% RSLogix 500 project FIVE_CONVEYER_SYS_BAK010.RSS, saved by version 8.30.00.16 %
PROJECT "UNTITLED"    % processor: Bul.1763 MicroLogix 1100 Series B %

PROGRAM FILES
  LAD 2   11 rungs
  LAD 3 "BELT 1"  5 rungs
  LAD 4 "BELT 2"  5 rungs
  LAD 5 "BELT 3"  5 rungs
  LAD 6 "BELT 4"  5 rungs
  LAD 7 "BELT 5"  5 rungs
  LAD 8 "SEQUENCING"  7 rungs

DATA FILES
  O0 OUTPUT  4 elements
  I1 INPUT  6 elements
  S2 STATUS  66 elements
  B3 BINARY  10 elements
  T4 TIMER  20 elements
  C5 COUNTER  1 elements
  R6 CONTROL  1 elements
  N7 INTEGER  1 elements
  F8 FLOAT  1 elements

LADDER 2
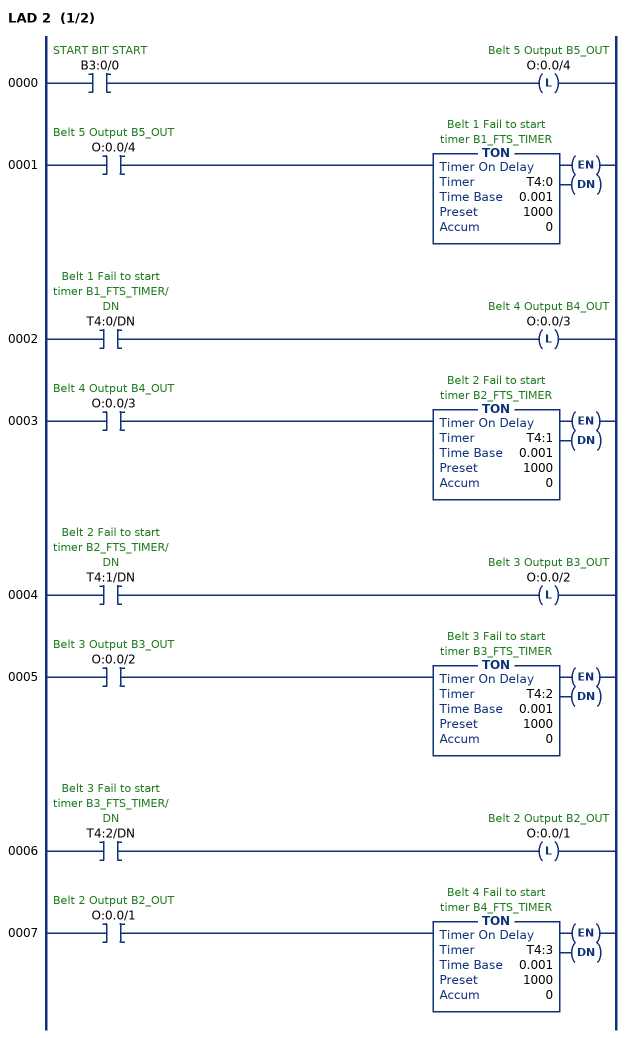
% Rung: 0 %  % edit flag set %
SOR XIC B3:0/0 OTL O:0.0/4 EOR
%   B3:0/0  START  "START BIT" %
%   O:0.0/4  B5_OUT  "Belt 5 Output" %
% Rung: 1 %  % edit flag set %
SOR XIC O:0.0/4 TON T4:0 0.001 1000 0 EOR
%   O:0.0/4  B5_OUT  "Belt 5 Output" %
%   T4:0  B1_FTS_TIMER  "Belt 1 Fail to start timer" %
% Rung: 2 %  % edit flag set %
SOR XIC T4:0/DN OTL O:0.0/3 EOR
%   T4:0  B1_FTS_TIMER  "Belt 1 Fail to start timer" %
%   O:0.0/3  B4_OUT  "Belt 4 Output" %
% Rung: 3 %  % edit flag set %
SOR XIC O:0.0/3 TON T4:1 0.001 1000 0 EOR
%   O:0.0/3  B4_OUT  "Belt 4 Output" %
%   T4:1  B2_FTS_TIMER  "Belt 2 Fail to start timer" %
% Rung: 4 %  % edit flag set %
SOR XIC T4:1/DN OTL O:0.0/2 EOR
%   T4:1  B2_FTS_TIMER  "Belt 2 Fail to start timer" %
%   O:0.0/2  B3_OUT  "Belt 3 Output" %
% Rung: 5 %  % edit flag set %
SOR XIC O:0.0/2 TON T4:2 0.001 1000 0 EOR
%   O:0.0/2  B3_OUT  "Belt 3 Output" %
%   T4:2  B3_FTS_TIMER  "Belt 3 Fail to start timer" %
% Rung: 6 %  % edit flag set %
SOR XIC T4:2/DN OTL O:0.0/1 EOR
%   T4:2  B3_FTS_TIMER  "Belt 3 Fail to start timer" %
%   O:0.0/1  B2_OUT  "Belt 2 Output" %
% Rung: 7 %  % edit flag set %
SOR XIC O:0.0/1 TON T4:3 0.001 1000 0 EOR
%   O:0.0/1  B2_OUT  "Belt 2 Output" %
%   T4:3  B4_FTS_TIMER  "Belt 4 Fail to start timer" %

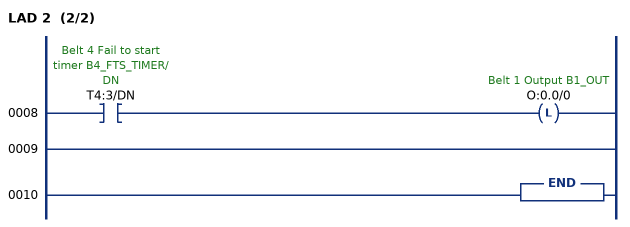
% Rung: 8 %  % edit flag set %
SOR XIC T4:3/DN OTL O:0.0/0 EOR
%   T4:3  B4_FTS_TIMER  "Belt 4 Fail to start timer" %
%   O:0.0/0  B1_OUT  "Belt 1 Output" %
% Rung: 9 %  % edit flag set %
SOR EOR
% Rung: 10 %
SOR END EOR

LADDER 3 "BELT 1"
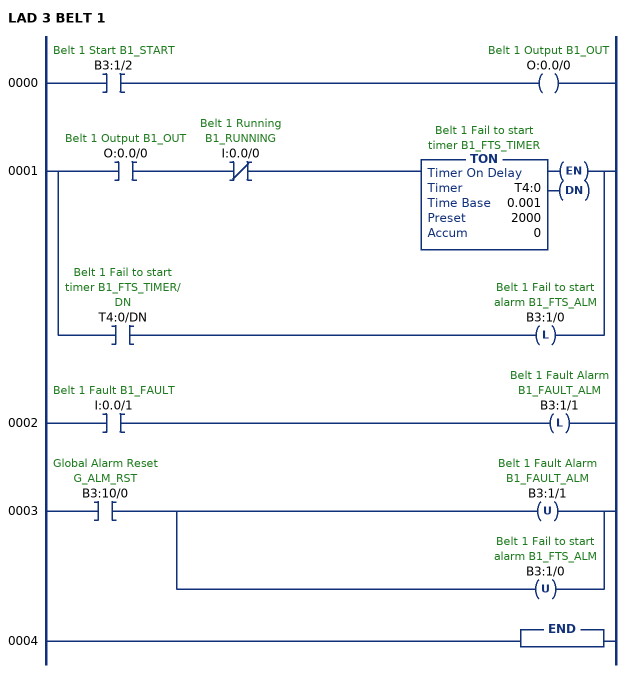
% Rung: 0 %  % edit flag set %
SOR XIC B3:1/2 OTE O:0.0/0 EOR
%   B3:1/2  B1_START  "Belt 1 Start" %
%   O:0.0/0  B1_OUT  "Belt 1 Output" %
% Rung: 1 %  % edit flag set %
SOR BST XIC O:0.0/0 XIO I:0.0/0 TON T4:0 0.001 2000 0 NXB XIC T4:0/DN OTL B3:1/0 BND EOR
%   O:0.0/0  B1_OUT  "Belt 1 Output" %
%   I:0.0/0  B1_RUNNING  "Belt 1 Running" %
%   T4:0  B1_FTS_TIMER  "Belt 1 Fail to start timer" %
%   B3:1/0  B1_FTS_ALM  "Belt 1 Fail to start alarm" %
% Rung: 2 %  % edit flag set %
SOR XIC I:0.0/1 OTL B3:1/1 EOR
%   I:0.0/1  B1_FAULT  "Belt 1 Fault" %
%   B3:1/1  B1_FAULT_ALM  "Belt 1 Fault Alarm" %
% Rung: 3 %  % edit flag set %
SOR XIC B3:10/0 BST OTU B3:1/1 NXB OTU B3:1/0 BND EOR
%   B3:10/0  G_ALM_RST  "Global Alarm Reset" %
%   B3:1/1  B1_FAULT_ALM  "Belt 1 Fault Alarm" %
%   B3:1/0  B1_FTS_ALM  "Belt 1 Fail to start alarm" %
% Rung: 4 %
SOR END EOR

LADDER 4 "BELT 2"
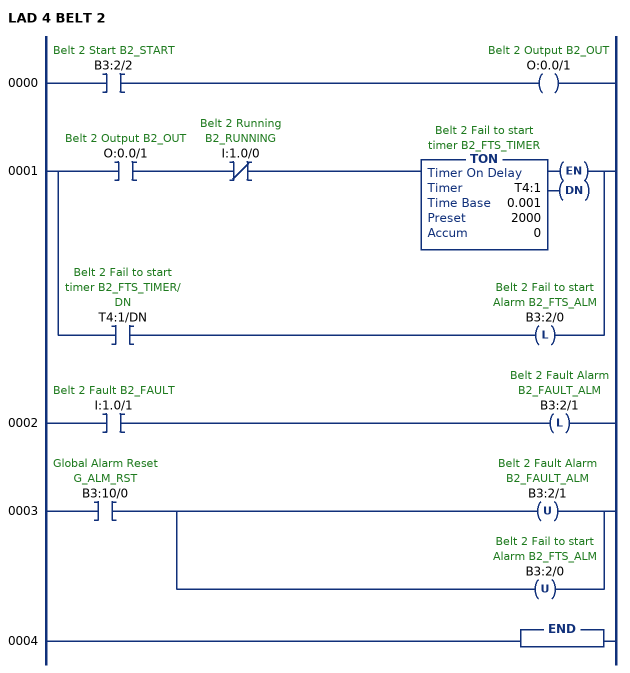
% Rung: 0 %  % edit flag set %
SOR XIC B3:2/2 OTE O:0.0/1 EOR
%   B3:2/2  B2_START  "Belt 2 Start" %
%   O:0.0/1  B2_OUT  "Belt 2 Output" %
% Rung: 1 %  % edit flag set %
SOR BST XIC O:0.0/1 XIO I:1.0/0 TON T4:1 0.001 2000 0 NXB XIC T4:1/DN OTL B3:2/0 BND EOR
%   O:0.0/1  B2_OUT  "Belt 2 Output" %
%   I:1.0/0  B2_RUNNING  "Belt 2 Running" %
%   T4:1  B2_FTS_TIMER  "Belt 2 Fail to start timer" %
%   B3:2/0  B2_FTS_ALM  "Belt 2 Fail to start Alarm" %
% Rung: 2 %  % edit flag set %
SOR XIC I:1.0/1 OTL B3:2/1 EOR
%   I:1.0/1  B2_FAULT  "Belt 2 Fault" %
%   B3:2/1  B2_FAULT_ALM  "Belt 2 Fault Alarm" %
% Rung: 3 %  % edit flag set %
SOR XIC B3:10/0 BST OTU B3:2/1 NXB OTU B3:2/0 BND EOR
%   B3:10/0  G_ALM_RST  "Global Alarm Reset" %
%   B3:2/1  B2_FAULT_ALM  "Belt 2 Fault Alarm" %
%   B3:2/0  B2_FTS_ALM  "Belt 2 Fail to start Alarm" %
% Rung: 4 %
SOR END EOR

LADDER 5 "BELT 3"
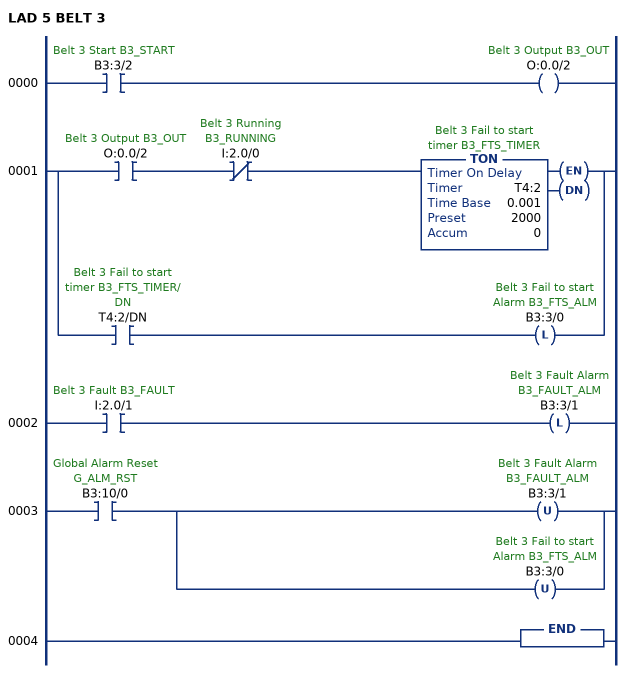
% Rung: 0 %  % edit flag set %
SOR XIC B3:3/2 OTE O:0.0/2 EOR
%   B3:3/2  B3_START  "Belt 3 Start" %
%   O:0.0/2  B3_OUT  "Belt 3 Output" %
% Rung: 1 %  % edit flag set %
SOR BST XIC O:0.0/2 XIO I:2.0/0 TON T4:2 0.001 2000 0 NXB XIC T4:2/DN OTL B3:3/0 BND EOR
%   O:0.0/2  B3_OUT  "Belt 3 Output" %
%   I:2.0/0  B3_RUNNING  "Belt 3 Running" %
%   T4:2  B3_FTS_TIMER  "Belt 3 Fail to start timer" %
%   B3:3/0  B3_FTS_ALM  "Belt 3 Fail to start Alarm" %
% Rung: 2 %  % edit flag set %
SOR XIC I:2.0/1 OTL B3:3/1 EOR
%   I:2.0/1  B3_FAULT  "Belt 3 Fault" %
%   B3:3/1  B3_FAULT_ALM  "Belt 3 Fault Alarm" %
% Rung: 3 %  % edit flag set %
SOR XIC B3:10/0 BST OTU B3:3/1 NXB OTU B3:3/0 BND EOR
%   B3:10/0  G_ALM_RST  "Global Alarm Reset" %
%   B3:3/1  B3_FAULT_ALM  "Belt 3 Fault Alarm" %
%   B3:3/0  B3_FTS_ALM  "Belt 3 Fail to start Alarm" %
% Rung: 4 %
SOR END EOR

LADDER 6 "BELT 4"
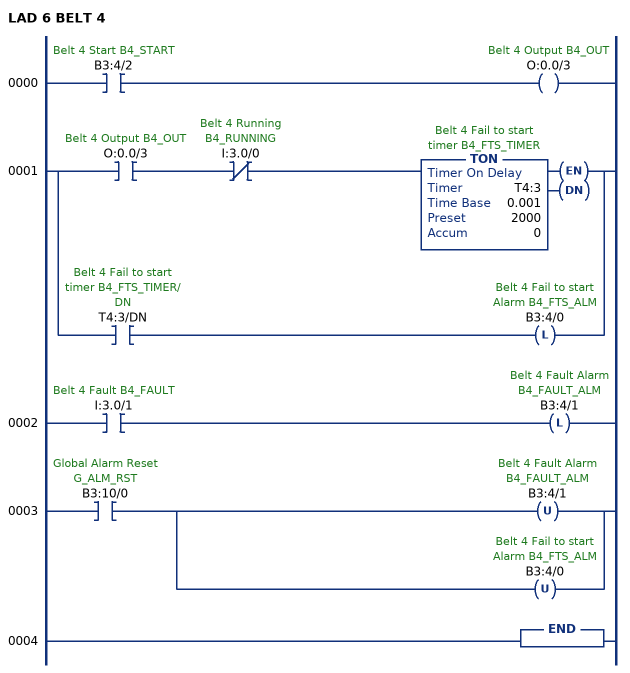
% Rung: 0 %  % edit flag set %
SOR XIC B3:4/2 OTE O:0.0/3 EOR
%   B3:4/2  B4_START  "Belt 4 Start" %
%   O:0.0/3  B4_OUT  "Belt 4 Output" %
% Rung: 1 %  % edit flag set %
SOR BST XIC O:0.0/3 XIO I:3.0/0 TON T4:3 0.001 2000 0 NXB XIC T4:3/DN OTL B3:4/0 BND EOR
%   O:0.0/3  B4_OUT  "Belt 4 Output" %
%   I:3.0/0  B4_RUNNING  "Belt 4 Running" %
%   T4:3  B4_FTS_TIMER  "Belt 4 Fail to start timer" %
%   B3:4/0  B4_FTS_ALM  "Belt 4 Fail to start Alarm" %
% Rung: 2 %  % edit flag set %
SOR XIC I:3.0/1 OTL B3:4/1 EOR
%   I:3.0/1  B4_FAULT  "Belt 4 Fault" %
%   B3:4/1  B4_FAULT_ALM  "Belt 4 Fault Alarm" %
% Rung: 3 %  % edit flag set %
SOR XIC B3:10/0 BST OTU B3:4/1 NXB OTU B3:4/0 BND EOR
%   B3:10/0  G_ALM_RST  "Global Alarm Reset" %
%   B3:4/1  B4_FAULT_ALM  "Belt 4 Fault Alarm" %
%   B3:4/0  B4_FTS_ALM  "Belt 4 Fail to start Alarm" %
% Rung: 4 %
SOR END EOR

LADDER 7 "BELT 5"
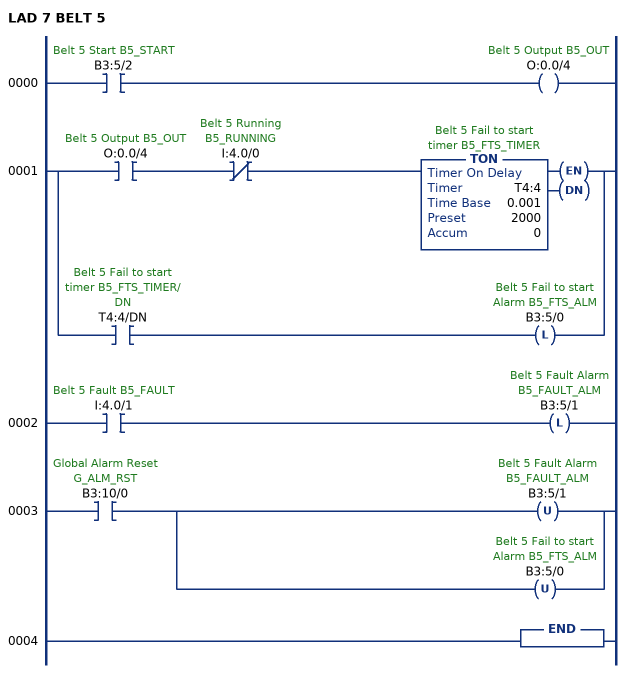
% Rung: 0 %  % edit flag set %
SOR XIC B3:5/2 OTE O:0.0/4 EOR
%   B3:5/2  B5_START  "Belt 5 Start" %
%   O:0.0/4  B5_OUT  "Belt 5 Output" %
% Rung: 1 %  % edit flag set %
SOR BST XIC O:0.0/4 XIO I:4.0/0 TON T4:4 0.001 2000 0 NXB XIC T4:4/DN OTL B3:5/0 BND EOR
%   O:0.0/4  B5_OUT  "Belt 5 Output" %
%   I:4.0/0  B5_RUNNING  "Belt 5 Running" %
%   T4:4  B5_FTS_TIMER  "Belt 5 Fail to start timer" %
%   B3:5/0  B5_FTS_ALM  "Belt 5 Fail to start Alarm" %
% Rung: 2 %  % edit flag set %
SOR XIC I:4.0/1 OTL B3:5/1 EOR
%   I:4.0/1  B5_FAULT  "Belt 5 Fault" %
%   B3:5/1  B5_FAULT_ALM  "Belt 5 Fault Alarm" %
% Rung: 3 %  % edit flag set %
SOR XIC B3:10/0 BST OTU B3:5/1 NXB OTU B3:5/0 BND EOR
%   B3:10/0  G_ALM_RST  "Global Alarm Reset" %
%   B3:5/1  B5_FAULT_ALM  "Belt 5 Fault Alarm" %
%   B3:5/0  B5_FTS_ALM  "Belt 5 Fail to start Alarm" %
% Rung: 4 %
SOR END EOR

LADDER 8 "SEQUENCING"
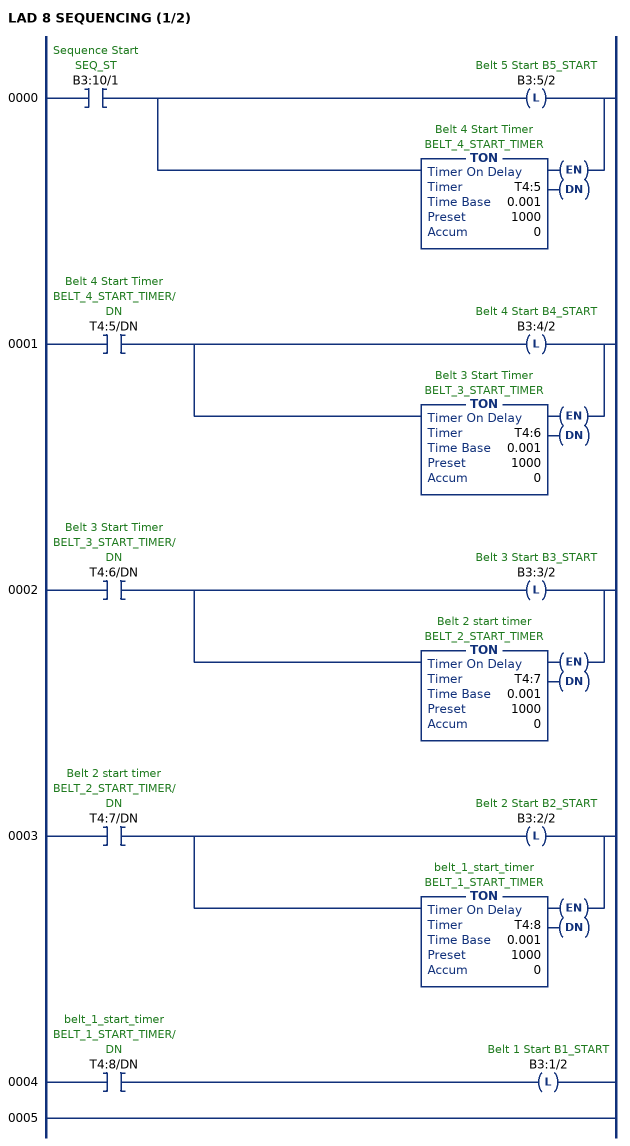
% Rung: 0 %  % edit flag set %
SOR XIC B3:10/1 BST OTL B3:5/2 NXB TON T4:5 0.001 1000 0 BND EOR
%   B3:10/1  SEQ_ST  "Sequence Start" %
%   B3:5/2  B5_START  "Belt 5 Start" %
%   T4:5  BELT_4_START_TIMER  "Belt 4 Start Timer" %
% Rung: 1 %  % edit flag set %
SOR XIC T4:5/DN BST OTL B3:4/2 NXB TON T4:6 0.001 1000 0 BND EOR
%   T4:5  BELT_4_START_TIMER  "Belt 4 Start Timer" %
%   B3:4/2  B4_START  "Belt 4 Start" %
%   T4:6  BELT_3_START_TIMER  "Belt 3 Start Timer" %
% Rung: 2 %  % edit flag set %
SOR XIC T4:6/DN BST OTL B3:3/2 NXB TON T4:7 0.001 1000 0 BND EOR
%   T4:6  BELT_3_START_TIMER  "Belt 3 Start Timer" %
%   B3:3/2  B3_START  "Belt 3 Start" %
%   T4:7  BELT_2_START_TIMER  "Belt 2 start timer" %
% Rung: 3 %  % edit flag set %
SOR XIC T4:7/DN BST OTL B3:2/2 NXB TON T4:8 0.001 1000 0 BND EOR
%   T4:7  BELT_2_START_TIMER  "Belt 2 start timer" %
%   B3:2/2  B2_START  "Belt 2 Start" %
%   T4:8  BELT_1_START_TIMER  "belt_1_start_timer" %
% Rung: 4 %  % edit flag set %
SOR XIC T4:8/DN OTL B3:1/2 EOR
%   T4:8  BELT_1_START_TIMER  "belt_1_start_timer" %
%   B3:1/2  B1_START  "Belt 1 Start" %
% Rung: 5 %  % edit flag set %
SOR EOR

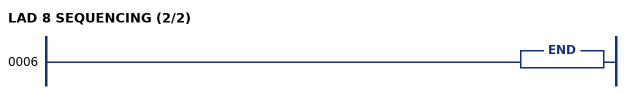
% Rung: 6 %
SOR END EOR

OTHER DOCUMENTED ADDRESSES
    "Belt 2 Fail to start timer"
  T4:0/5  B4_START_TIMER  "Belt 4 Start Timer"
  T4:6.ACC  "Belt 3 Start Timer"

DATA TABLE (non-zero values as saved)
DATA T4
% .PRE .ACC %
% T4:0 % 1000 0
% T4:1 % 1000 0
% T4:2 % 1000 0
% T4:3 % 1000 0
